{attribute 'qualified_only'}
{attribute 'strict'}
TYPE EBehaviorType :
(
	none := 0,
	control_primitive := 1,
	user_sequence := 2,
	generated_sequence := 3
);
END_TYPE

(* stored: Version 1.1.0.1, ProductVersion 3.1.4024.9
   DUT EBehaviorType: Id {6d6df99a-b2b8-4a24-912d-cfd76aec06e4} *)
